Staubli VAL3: isIDAvailable.pgx

public program isIDAvailable(num& x_nCamID (dimensions=1), bool& x_bError (dimensions=1))
begin
  //-----------------------------------------------------------------------
  //Header begin
  //Description of program
  //  Verify wether an ID is available or not.
  //Input parameters :
  //  num x_nCamID :
  //    role: ID to check the availability of
  //Output parameters
  //  bool x_bError :
  //    role : true if x_nCamID available, false otherwise
  //
  //Examples
  //    call isIDAvailable(l_nCamID,l_bError)
  //
  //History
  //  Creation : 25-05-12 - t.caille - c.rocchini
  //Header end
  //-----------------------------------------------------------------------
  if x_nCamID<size(cCamera)-1 and cCamera[x_nCamID].bConnected==false
    x_bError=false
  else
    x_bError=true
    nLibErrorCode=200
  endIf
end
